TYPE
    TcoPlrPaletizator_Status_v_1_x_x EXTENDS TcoFeeding_Status_v_1_x_x:
    STRUCT

        
		EntryBufferEmpty:BOOL;
        BlisterReady : BOOL;
        OutBufferFull : BOOL;
    END_STRUCT
END_TYPE

(* stored: Version 1.1.0.1
   DUT TcoPlrPaletizator_Status_v_1_x_x: Id {63863fed-97a2-49c5-91a5-46ab30ebc9cd} *)
